// TIA Portal project "APD Gateway Customer Library Source v02_01_00" (V17)
// 00.00.01 - integrated tag tables
// 02.00.01 - v2 will have flat entrypoint
// 02.00.02 - poke ip flattened, next up: finish system parameters
// 02.00.03 - sign formats
// 02.00.04 - line formats
// 02.00.05 - segment formats
// 02.01.00 - released v2

(* hardware
DEVICE "S7-1200 station_1"  S7-1200 Station
   slot 0: "Rack_0"  S7-1200 Rack  Rack  V1.0
   slot 1: "interfacelibrary"  CPU 1215C AC/DC/Rly  6ES7 215-1BG40-0XB0  V4.0
DEVICE "GSD device_1"  GSD.Device.PN
   slot 0: "Rack"  Rack  V1.0
   slot 1: "adpgateway"  Profinet_to_ADP_Gateway  6ES7 212-1AE40-0XB0  V4.5
      slot 0: "Message"  Message
      slot 1: "Interface"  Interface
         slot 1: "Port 1"  Port 1
*)

// ===== PLC "interfacelibrary"  CPU 1215C AC/DC/Rly =====

VAR_GLOBAL   // PLC tag table "Default tag table"
   "System_Byte" AT %MB1 : Byte;
   "FirstScan" AT %M1.0 : Bool;
   "DiagStatusUpdate" AT %M1.1 : Bool;
   "AlwaysTRUE" AT %M1.2 : Bool;
   "AlwaysFALSE" AT %M1.3 : Bool;
   "Clock_Byte" AT %MB0 : Byte;
   "Clock_10Hz" AT %M0.0 : Bool;
   "Clock_5Hz" AT %M0.1 : Bool;
   "Clock_2.5Hz" AT %M0.2 : Bool;
   "Clock_2Hz" AT %M0.3 : Bool;
   "Clock_1.25Hz" AT %M0.4 : Bool;
   "Clock_1Hz" AT %M0.5 : Bool;
   "Clock_0.625Hz" AT %M0.6 : Bool;
   "Clock_0.5Hz" AT %M0.7 : Bool;
END_VAR

VAR_GLOBAL   // PLC tag table "Line Format"
   "Line_0_Font_Size_&_Weight" AT %QB20 : USInt;
   "Line_0_Horizontal_Alignment" AT %QB21 : USInt;
   "Line_1_Font_Size_&_Weight" AT %QB22 : USInt;
   "Line_1_Horizontal_Alignment" AT %QB23 : USInt;
   "Line_2_Font_Size_&_Weight" AT %QB24 : USInt;
   "Line_2_Horizontal_Alignment" AT %QB25 : USInt;
   "Line_3_Font_Size_&_Weight" AT %QB26 : USInt;
   "Line_3_Horizontal_Alignment" AT %QB27 : USInt;
   "Line_4_Font_Size_&_Weight" AT %QB28 : USInt;
   "Line_4_Horizontal_Alignment" AT %QB29 : USInt;
END_VAR

VAR_GLOBAL   // PLC tag table "Segment Format 0"
   "Segment_Format_0_FG_Color" AT %QB50 : SInt;
   "Segment_Format_0_BG_Color" AT %QB51 : SInt;
   "Segment_Format_0_Flash" AT %QB52 : SInt;
   "Segment_Format_0_Line_Number" AT %QB53 : SInt;
   "Segment_Format_0_Text_Byte_0" AT %QB54 : Char;
   "Segment_Format_0_Text_Byte_1" AT %QB55 : Char;
   "Segment_Format_0_Text_Byte_2" AT %QB56 : Char;
   "Segment_Format_0_Text_Byte_3" AT %QB57 : Char;
   "Segment_Format_0_Text_Byte_4" AT %QB58 : Char;
   "Segment_Format_0_Text_Byte_5" AT %QB59 : Char;
   "Segment_Format_0_Text_Byte_6" AT %QB60 : Char;
   "Segment_Format_0_Text_Byte_7" AT %QB61 : Char;
   "Segment_Format_0_Text_Byte_8" AT %QB62 : Char;
   "Segment_Format_0_Text_Byte_9" AT %QB63 : Char;
   "Segment_Format_0_Text_Byte_10" AT %QB64 : Char;
   "Segment_Format_0_Text_Byte_11" AT %QB65 : Char;
   "Segment_Format_0_Text_Byte_12" AT %QB66 : Char;
   "Segment_Format_0_Text_Byte_13" AT %QB67 : Char;
   "Segment_Format_0_Text_Byte_14" AT %QB68 : Char;
   "Segment_Format_0_Text_Byte_15" AT %QB69 : Char;
   "Segment_Format_0_Text_Byte_16" AT %QB70 : Char;
   "Segment_Format_0_Text_Byte_17" AT %QB71 : Char;
   "Segment_Format_0_Text_Byte_18" AT %QB72 : Char;
   "Segment_Format_0_Text_Byte_19" AT %QB73 : Char;
   "Segment_Format_0_Text_Byte_20" AT %QB74 : Char;
   "Segment_Format_0_Text_Byte_21" AT %QB75 : Char;
   "Segment_Format_0_Text_Byte_22" AT %QB76 : Char;
   "Segment_Format_0_Text_Byte_23" AT %QB77 : Char;
   "Segment_Format_0_Text_Byte_24" AT %QB78 : Char;
   "Segment_Format_0_Text_Byte_25" AT %QB79 : Char;
   "Segment_Format_0_Text_Byte_26" AT %QB80 : Char;
   "Segment_Format_0_Text_Byte_27" AT %QB81 : Char;
   "Segment_Format_0_Text_Byte_28" AT %QB82 : Char;
   "Segment_Format_0_Text_Byte_29" AT %QB83 : Char;
   "Segment_Format_0_Text_Byte_30" AT %QB84 : Char;
   "Segment_Format_0_Text_Byte_31" AT %QB85 : Char;
   "Segment_Format_0_Text_Byte_32" AT %QB86 : Char;
   "Segment_Format_0_Text_Byte_33" AT %QB87 : Char;
   "Segment_Format_0_Text_Byte_34" AT %QB88 : Char;
   "Segment_Format_0_Text_Byte_35" AT %QB89 : Char;
   "Segment_Format_0_Text_Byte_36" AT %QB90 : Char;
   "Segment_Format_0_Text_Byte_37" AT %QB91 : Char;
   "Segment_Format_0_Text_Byte_38" AT %QB92 : Char;
   "Segment_Format_0_Text_Byte_39" AT %QB93 : Char;
   "Segment_Format_0_Text_Byte_40" AT %QB94 : Char;
   "Segment_Format_0_Text_Byte_41" AT %QB95 : Char;
   "Segment_Format_0_Text_Byte_42" AT %QB96 : Char;
   "Segment_Format_0_Text_Byte_43" AT %QB97 : Char;
   "Segment_Format_0_Text_Byte_44" AT %QB98 : Char;
   "Segment_Format_0_Text_Byte_45" AT %QB99 : Char;
END_VAR

VAR_GLOBAL   // PLC tag table "Segment Format 1"
   "Segment_Format_1_FG_Color" AT %QB100 : USInt;
   "Segment_Format_1_BG_Color" AT %QB101 : USInt;
   "Segment_Format_1_Flash" AT %QB102 : USInt;
   "Segment_Format_1_Line_Number" AT %QB103 : USInt;
   "Segment_Format_1_Text_Byte_0" AT %QB104 : Char;
   "Segment_Format_1_Text_Byte_1" AT %QB105 : Char;
   "Segment_Format_1_Text_Byte_2" AT %QB106 : Char;
   "Segment_Format_1_Text_Byte_3" AT %QB107 : Char;
   "Segment_Format_1_Text_Byte_4" AT %QB108 : Char;
   "Segment_Format_1_Text_Byte_5" AT %QB109 : Char;
   "Segment_Format_1_Text_Byte_6" AT %QB110 : Char;
   "Segment_Format_1_Text_Byte_7" AT %QB111 : Char;
   "Segment_Format_1_Text_Byte_8" AT %QB112 : Char;
   "Segment_Format_1_Text_Byte_9" AT %QB113 : Char;
   "Segment_Format_1_Text_Byte_10" AT %QB114 : Char;
   "Segment_Format_1_Text_Byte_11" AT %QB115 : Char;
   "Segment_Format_1_Text_Byte_12" AT %QB116 : Char;
   "Segment_Format_1_Text_Byte_13" AT %QB117 : Char;
   "Segment_Format_1_Text_Byte_14" AT %QB118 : Char;
   "Segment_Format_1_Text_Byte_15" AT %QB119 : Char;
   "Segment_Format_1_Text_Byte_16" AT %QB120 : Char;
   "Segment_Format_1_Text_Byte_17" AT %QB121 : Char;
   "Segment_Format_1_Text_Byte_18" AT %QB122 : Char;
   "Segment_Format_1_Text_Byte_19" AT %QB123 : Char;
   "Segment_Format_1_Text_Byte_20" AT %QB124 : Char;
   "Segment_Format_1_Text_Byte_21" AT %QB125 : Char;
   "Segment_Format_1_Text_Byte_22" AT %QB126 : Char;
   "Segment_Format_1_Text_Byte_23" AT %QB127 : Char;
   "Segment_Format_1_Text_Byte_24" AT %QB128 : Char;
   "Segment_Format_1_Text_Byte_25" AT %QB129 : Char;
   "Segment_Format_1_Text_Byte_26" AT %QB130 : Char;
   "Segment_Format_1_Text_Byte_27" AT %QB131 : Char;
   "Segment_Format_1_Text_Byte_28" AT %QB132 : Char;
   "Segment_Format_1_Text_Byte_29" AT %QB133 : Char;
   "Segment_Format_1_Text_Byte_30" AT %QB134 : Char;
   "Segment_Format_1_Text_Byte_31" AT %QB135 : Char;
   "Segment_Format_1_Text_Byte_32" AT %QB136 : Char;
   "Segment_Format_1_Text_Byte_33" AT %QB137 : Char;
   "Segment_Format_1_Text_Byte_34" AT %QB138 : Char;
   "Segment_Format_1_Text_Byte_35" AT %QB139 : Char;
   "Segment_Format_1_Text_Byte_36" AT %QB140 : Char;
   "Segment_Format_1_Text_Byte_37" AT %QB141 : Char;
   "Segment_Format_1_Text_Byte_38" AT %QB142 : Char;
   "Segment_Format_1_Text_Byte_39" AT %QB143 : Char;
   "Segment_Format_1_Text_Byte_40" AT %QB144 : Char;
   "Segment_Format_1_Text_Byte_41" AT %QB145 : Char;
   "Segment_Format_1_Text_Byte_42" AT %QB146 : Char;
   "Segment_Format_1_Text_Byte_43" AT %QB147 : Char;
   "Segment_Format_1_Text_Byte_44" AT %QB148 : Char;
   "Segment_Format_1_Text_Byte_45" AT %QB149 : Char;
END_VAR

VAR_GLOBAL   // PLC tag table "Segment Format 2"
   "Segment_Format_2_FG_Color" AT %QB150 : USInt;
   "Segment_Format_2_BG_Color" AT %QB151 : USInt;
   "Segment_Format_2_Flash" AT %QB152 : USInt;
   "Segment_Format_2_Line_Number" AT %QB153 : USInt;
   "Segment_Format_2_Text_Byte_0" AT %QB154 : Char;
   "Segment_Format_2_Text_Byte_1" AT %QB155 : Char;
   "Segment_Format_2_Text_Byte_2" AT %QB156 : Char;
   "Segment_Format_2_Text_Byte_3" AT %QB157 : Char;
   "Segment_Format_2_Text_Byte_4" AT %QB158 : Char;
   "Segment_Format_2_Text_Byte_5" AT %QB159 : Char;
   "Segment_Format_2_Text_Byte_6" AT %QB160 : Char;
   "Segment_Format_2_Text_Byte_7" AT %QB161 : Char;
   "Segment_Format_2_Text_Byte_8" AT %QB162 : Char;
   "Segment_Format_2_Text_Byte_9" AT %QB163 : Char;
   "Segment_Format_2_Text_Byte_10" AT %QB164 : Char;
   "Segment_Format_2_Text_Byte_11" AT %QB165 : Char;
   "Segment_Format_2_Text_Byte_12" AT %QB166 : Char;
   "Segment_Format_2_Text_Byte_13" AT %QB167 : Char;
   "Segment_Format_2_Text_Byte_14" AT %QB168 : Char;
   "Segment_Format_2_Text_Byte_15" AT %QB169 : Char;
   "Segment_Format_2_Text_Byte_16" AT %QB170 : Char;
   "Segment_Format_2_Text_Byte_17" AT %QB171 : Char;
   "Segment_Format_2_Text_Byte_18" AT %QB172 : Char;
   "Segment_Format_2_Text_Byte_19" AT %QB173 : Char;
   "Segment_Format_2_Text_Byte_20" AT %QB174 : Char;
   "Segment_Format_2_Text_Byte_21" AT %QB175 : Char;
   "Segment_Format_2_Text_Byte_22" AT %QB176 : Char;
   "Segment_Format_2_Text_Byte_23" AT %QB177 : Char;
   "Segment_Format_2_Text_Byte_24" AT %QB178 : Char;
   "Segment_Format_2_Text_Byte_25" AT %QB179 : Char;
   "Segment_Format_2_Text_Byte_26" AT %QB180 : Char;
   "Segment_Format_2_Text_Byte_27" AT %QB181 : Char;
   "Segment_Format_2_Text_Byte_28" AT %QB182 : Char;
   "Segment_Format_2_Text_Byte_29" AT %QB183 : Char;
   "Segment_Format_2_Text_Byte_30" AT %QB184 : Char;
   "Segment_Format_2_Text_Byte_31" AT %QB185 : Char;
   "Segment_Format_2_Text_Byte_32" AT %QB186 : Char;
   "Segment_Format_2_Text_Byte_33" AT %QB187 : Char;
   "Segment_Format_2_Text_Byte_34" AT %QB188 : Char;
   "Segment_Format_2_Text_Byte_35" AT %QB189 : Char;
   "Segment_Format_2_Text_Byte_36" AT %QB190 : Char;
   "Segment_Format_2_Text_Byte_37" AT %QB191 : Char;
   "Segment_Format_2_Text_Byte_38" AT %QB192 : Char;
   "Segment_Format_2_Text_Byte_39" AT %QB193 : Char;
   "Segment_Format_2_Text_Byte_40" AT %QB194 : Char;
   "Segment_Format_2_Text_Byte_41" AT %QB195 : Char;
   "Segment_Format_2_Text_Byte_42" AT %QB196 : Char;
   "Segment_Format_2_Text_Byte_43" AT %QB197 : Char;
   "Segment_Format_2_Text_Byte_44" AT %QB198 : Char;
   "Segment_Format_2_Text_Byte_45" AT %QB199 : Char;
END_VAR

VAR_GLOBAL   // PLC tag table "Segment Format 3"
   "Segment_Format_3_FG_Color" AT %QB200 : USInt;
   "Segment_Format_3_BG_Color" AT %QB201 : USInt;
   "Segment_Format_3_Flash" AT %QB202 : USInt;
   "Segment_Format_3_Line_Number" AT %QB203 : USInt;
   "Segment_Format_3_Text_Byte_0" AT %QB204 : Char;
   "Segment_Format_3_Text_Byte_1" AT %QB205 : Char;
   "Segment_Format_3_Text_Byte_2" AT %QB206 : Char;
   "Segment_Format_3_Text_Byte_3" AT %QB207 : Char;
   "Segment_Format_3_Text_Byte_4" AT %QB208 : Char;
   "Segment_Format_3_Text_Byte_5" AT %QB209 : Char;
   "Segment_Format_3_Text_Byte_6" AT %QB210 : Char;
   "Segment_Format_3_Text_Byte_7" AT %QB211 : Char;
   "Segment_Format_3_Text_Byte_8" AT %QB212 : Char;
   "Segment_Format_3_Text_Byte_9" AT %QB213 : Char;
   "Segment_Format_3_Text_Byte_10" AT %QB214 : Char;
   "Segment_Format_3_Text_Byte_11" AT %QB215 : Char;
   "Segment_Format_3_Text_Byte_12" AT %QB216 : Char;
   "Segment_Format_3_Text_Byte_13" AT %QB217 : Char;
   "Segment_Format_3_Text_Byte_14" AT %QB218 : Char;
   "Segment_Format_3_Text_Byte_15" AT %QB219 : Char;
   "Segment_Format_3_Text_Byte_16" AT %QB220 : Char;
   "Segment_Format_3_Text_Byte_17" AT %QB221 : Char;
   "Segment_Format_3_Text_Byte_18" AT %QB222 : Char;
   "Segment_Format_3_Text_Byte_19" AT %QB223 : Char;
   "Segment_Format_3_Text_Byte_20" AT %QB224 : Char;
   "Segment_Format_3_Text_Byte_21" AT %QB225 : Char;
   "Segment_Format_3_Text_Byte_22" AT %QB226 : Char;
   "Segment_Format_3_Text_Byte_23" AT %QB227 : Char;
   "Segment_Format_3_Text_Byte_24" AT %QB228 : Char;
   "Segment_Format_3_Text_Byte_25" AT %QB229 : Char;
   "Segment_Format_3_Text_Byte_26" AT %QB230 : Char;
   "Segment_Format_3_Text_Byte_27" AT %QB231 : Char;
   "Segment_Format_3_Text_Byte_28" AT %QB232 : Char;
   "Segment_Format_3_Text_Byte_29" AT %QB233 : Char;
   "Segment_Format_3_Text_Byte_30" AT %QB234 : Char;
   "Segment_Format_3_Text_Byte_31" AT %QB235 : Char;
   "Segment_Format_3_Text_Byte_32" AT %QB236 : Char;
   "Segment_Format_3_Text_Byte_33" AT %QB237 : Char;
   "Segment_Format_3_Text_Byte_34" AT %QB238 : Char;
   "Segment_Format_3_Text_Byte_35" AT %QB239 : Char;
   "Segment_Format_3_Text_Byte_36" AT %QB240 : Char;
   "Segment_Format_3_Text_Byte_37" AT %QB241 : Char;
   "Segment_Format_3_Text_Byte_38" AT %QB242 : Char;
   "Segment_Format_3_Text_Byte_39" AT %QB243 : Char;
   "Segment_Format_3_Text_Byte_40" AT %QB244 : Char;
   "Segment_Format_3_Text_Byte_41" AT %QB245 : Char;
   "Segment_Format_3_Text_Byte_42" AT %QB246 : Char;
   "Segment_Format_3_Text_Byte_43" AT %QB247 : Char;
   "Segment_Format_3_Text_Byte_44" AT %QB248 : Char;
   "Segment_Format_3_Text_Byte_45" AT %QB249 : Char;
END_VAR

VAR_GLOBAL   // PLC tag table "Segment Format 4"
   "Segment_Format_4_FG_Color" AT %QB250 : USInt;
   "Segment_Format_4_BG_Color" AT %QB251 : USInt;
   "Segment_Format_4_Flash" AT %QB252 : USInt;
   "Segment_Format_4_Line_Number" AT %QB253 : USInt;
   "Segment_Format_4_Text_Byte_0" AT %QB254 : Char;
   "Segment_Format_4_Text_Byte_1" AT %QB255 : Char;
   "Segment_Format_4_Text_Byte_2" AT %QB256 : Char;
   "Segment_Format_4_Text_Byte_3" AT %QB257 : Char;
   "Segment_Format_4_Text_Byte_4" AT %QB258 : Char;
   "Segment_Format_4_Text_Byte_5" AT %QB259 : Char;
   "Segment_Format_4_Text_Byte_6" AT %QB260 : Char;
   "Segment_Format_4_Text_Byte_7" AT %QB261 : Char;
   "Segment_Format_4_Text_Byte_8" AT %QB262 : Char;
   "Segment_Format_4_Text_Byte_9" AT %QB263 : Char;
   "Segment_Format_4_Text_Byte_10" AT %QB264 : Char;
   "Segment_Format_4_Text_Byte_11" AT %QB265 : Char;
   "Segment_Format_4_Text_Byte_12" AT %QB266 : Char;
   "Segment_Format_4_Text_Byte_13" AT %QB267 : Char;
   "Segment_Format_4_Text_Byte_14" AT %QB268 : Char;
   "Segment_Format_4_Text_Byte_15" AT %QB269 : Char;
   "Segment_Format_4_Text_Byte_16" AT %QB270 : Char;
   "Segment_Format_4_Text_Byte_17" AT %QB271 : Char;
   "Segment_Format_4_Text_Byte_18" AT %QB272 : Char;
   "Segment_Format_4_Text_Byte_19" AT %QB273 : Char;
   "Segment_Format_4_Text_Byte_20" AT %QB274 : Char;
   "Segment_Format_4_Text_Byte_21" AT %QB275 : Char;
   "Segment_Format_4_Text_Byte_22" AT %QB276 : Char;
   "Segment_Format_4_Text_Byte_23" AT %QB277 : Char;
   "Segment_Format_4_Text_Byte_24" AT %QB278 : Char;
   "Segment_Format_4_Text_Byte_25" AT %QB279 : Char;
   "Segment_Format_4_Text_Byte_26" AT %QB280 : Char;
   "Segment_Format_4_Text_Byte_27" AT %QB281 : Char;
   "Segment_Format_4_Text_Byte_28" AT %QB282 : Char;
   "Segment_Format_4_Text_Byte_29" AT %QB283 : Char;
   "Segment_Format_4_Text_Byte_30" AT %QB284 : Char;
   "Segment_Format_4_Text_Byte_31" AT %QB285 : Char;
   "Segment_Format_4_Text_Byte_32" AT %QB286 : Char;
   "Segment_Format_4_Text_Byte_33" AT %QB287 : Char;
   "Segment_Format_4_Text_Byte_34" AT %QB288 : Char;
   "Segment_Format_4_Text_Byte_35" AT %QB289 : Char;
   "Segment_Format_4_Text_Byte_36" AT %QB290 : Char;
   "Segment_Format_4_Text_Byte_37" AT %QB291 : Char;
   "Segment_Format_4_Text_Byte_38" AT %QB292 : Char;
   "Segment_Format_4_Text_Byte_39" AT %QB293 : Char;
   "Segment_Format_4_Text_Byte_40" AT %QB294 : Char;
   "Segment_Format_4_Text_Byte_41" AT %QB295 : Char;
   "Segment_Format_4_Text_Byte_42" AT %QB296 : Char;
   "Segment_Format_4_Text_Byte_43" AT %QB297 : Char;
   "Segment_Format_4_Text_Byte_44" AT %QB298 : Char;
   "Segment_Format_4_Text_Byte_45" AT %QB299 : Char;
END_VAR

VAR_GLOBAL   // PLC tag table "Segment Format 5"
   "Segment_Format_5_FG_Color" AT %QB300 : USInt;
   "Segment_Format_5_BG_Color" AT %QB301 : USInt;
   "Segment_Format_5_Flash" AT %QB302 : USInt;
   "Segment_Format_5_Line_Number" AT %QB303 : USInt;
   "Segment_Format_5_Text_Byte_0" AT %QB304 : Char;
   "Segment_Format_5_Text_Byte_1" AT %QB305 : Char;
   "Segment_Format_5_Text_Byte_2" AT %QB306 : Char;
   "Segment_Format_5_Text_Byte_3" AT %QB307 : Char;
   "Segment_Format_5_Text_Byte_4" AT %QB308 : Char;
   "Segment_Format_5_Text_Byte_5" AT %QB309 : Char;
   "Segment_Format_5_Text_Byte_6" AT %QB310 : Char;
   "Segment_Format_5_Text_Byte_7" AT %QB311 : Char;
   "Segment_Format_5_Text_Byte_8" AT %QB312 : Char;
   "Segment_Format_5_Text_Byte_9" AT %QB313 : Char;
   "Segment_Format_5_Text_Byte_10" AT %QB314 : Char;
   "Segment_Format_5_Text_Byte_11" AT %QB315 : Char;
   "Segment_Format_5_Text_Byte_12" AT %QB316 : Char;
   "Segment_Format_5_Text_Byte_13" AT %QB317 : Char;
   "Segment_Format_5_Text_Byte_14" AT %QB318 : Char;
   "Segment_Format_5_Text_Byte_15" AT %QB319 : Char;
   "Segment_Format_5_Text_Byte_16" AT %QB320 : Char;
   "Segment_Format_5_Text_Byte_17" AT %QB321 : Char;
   "Segment_Format_5_Text_Byte_18" AT %QB322 : Char;
   "Segment_Format_5_Text_Byte_19" AT %QB323 : Char;
   "Segment_Format_5_Text_Byte_20" AT %QB324 : Char;
   "Segment_Format_5_Text_Byte_21" AT %QB325 : Char;
   "Segment_Format_5_Text_Byte_22" AT %QB326 : Char;
   "Segment_Format_5_Text_Byte_23" AT %QB327 : Char;
   "Segment_Format_5_Text_Byte_24" AT %QB328 : Char;
   "Segment_Format_5_Text_Byte_25" AT %QB329 : Char;
   "Segment_Format_5_Text_Byte_26" AT %QB330 : Char;
   "Segment_Format_5_Text_Byte_27" AT %QB331 : Char;
   "Segment_Format_5_Text_Byte_28" AT %QB332 : Char;
   "Segment_Format_5_Text_Byte_29" AT %QB333 : Char;
   "Segment_Format_5_Text_Byte_30" AT %QB334 : Char;
   "Segment_Format_5_Text_Byte_31" AT %QB335 : Char;
   "Segment_Format_5_Text_Byte_32" AT %QB336 : Char;
   "Segment_Format_5_Text_Byte_33" AT %QB337 : Char;
   "Segment_Format_5_Text_Byte_34" AT %QB338 : Char;
   "Segment_Format_5_Text_Byte_35" AT %QB339 : Char;
   "Segment_Format_5_Text_Byte_36" AT %QB340 : Char;
   "Segment_Format_5_Text_Byte_37" AT %QB341 : Char;
   "Segment_Format_5_Text_Byte_38" AT %QB342 : Char;
   "Segment_Format_5_Text_Byte_39" AT %QB343 : Char;
   "Segment_Format_5_Text_Byte_40" AT %QB344 : Char;
   "Segment_Format_5_Text_Byte_41" AT %QB345 : Char;
   "Segment_Format_5_Text_Byte_42" AT %QB346 : Char;
   "Segment_Format_5_Text_Byte_43" AT %QB347 : Char;
   "Segment_Format_5_Text_Byte_44" AT %QB348 : Char;
   "Segment_Format_5_Text_Byte_45" AT %QB349 : Char;
END_VAR

VAR_GLOBAL   // PLC tag table "Segment Format 6"
   "Segment_Format_6_FG_Color" AT %QB350 : USInt;
   "Segment_Format_6_BG_Color" AT %QB351 : USInt;
   "Segment_Format_6_Flash" AT %QB352 : USInt;
   "Segment_Format_6_Line_Number" AT %QB353 : USInt;
   "Segment_Format_6_Text_Byte_0" AT %QB354 : Char;
   "Segment_Format_6_Text_Byte_1" AT %QB355 : Char;
   "Segment_Format_6_Text_Byte_2" AT %QB356 : Char;
   "Segment_Format_6_Text_Byte_3" AT %QB357 : Char;
   "Segment_Format_6_Text_Byte_4" AT %QB358 : Char;
   "Segment_Format_6_Text_Byte_5" AT %QB359 : Char;
   "Segment_Format_6_Text_Byte_6" AT %QB360 : Char;
   "Segment_Format_6_Text_Byte_7" AT %QB361 : Char;
   "Segment_Format_6_Text_Byte_8" AT %QB362 : Char;
   "Segment_Format_6_Text_Byte_9" AT %QB363 : Char;
   "Segment_Format_6_Text_Byte_10" AT %QB364 : Char;
   "Segment_Format_6_Text_Byte_11" AT %QB365 : Char;
   "Segment_Format_6_Text_Byte_12" AT %QB366 : Char;
   "Segment_Format_6_Text_Byte_13" AT %QB367 : Char;
   "Segment_Format_6_Text_Byte_14" AT %QB368 : Char;
   "Segment_Format_6_Text_Byte_15" AT %QB369 : Char;
   "Segment_Format_6_Text_Byte_16" AT %QB370 : Char;
   "Segment_Format_6_Text_Byte_17" AT %QB371 : Char;
   "Segment_Format_6_Text_Byte_18" AT %QB372 : Char;
   "Segment_Format_6_Text_Byte_19" AT %QB373 : Char;
   "Segment_Format_6_Text_Byte_20" AT %QB374 : Char;
   "Segment_Format_6_Text_Byte_21" AT %QB375 : Char;
   "Segment_Format_6_Text_Byte_22" AT %QB376 : Char;
   "Segment_Format_6_Text_Byte_23" AT %QB377 : Char;
   "Segment_Format_6_Text_Byte_24" AT %QB378 : Char;
   "Segment_Format_6_Text_Byte_25" AT %QB379 : Char;
   "Segment_Format_6_Text_Byte_26" AT %QB380 : Char;
   "Segment_Format_6_Text_Byte_27" AT %QB381 : Char;
   "Segment_Format_6_Text_Byte_28" AT %QB382 : Char;
   "Segment_Format_6_Text_Byte_29" AT %QB383 : Char;
   "Segment_Format_6_Text_Byte_30" AT %QB384 : Char;
   "Segment_Format_6_Text_Byte_31" AT %QB385 : Char;
   "Segment_Format_6_Text_Byte_32" AT %QB386 : Char;
   "Segment_Format_6_Text_Byte_33" AT %QB387 : Char;
   "Segment_Format_6_Text_Byte_34" AT %QB388 : Char;
   "Segment_Format_6_Text_Byte_35" AT %QB389 : Char;
   "Segment_Format_6_Text_Byte_36" AT %QB390 : Char;
   "Segment_Format_6_Text_Byte_37" AT %QB391 : Char;
   "Segment_Format_6_Text_Byte_38" AT %QB392 : Char;
   "Segment_Format_6_Text_Byte_39" AT %QB393 : Char;
   "Segment_Format_6_Text_Byte_40" AT %QB394 : Char;
   "Segment_Format_6_Text_Byte_41" AT %QB395 : Char;
   "Segment_Format_6_Text_Byte_42" AT %QB396 : Char;
   "Segment_Format_6_Text_Byte_43" AT %QB397 : Char;
   "Segment_Format_6_Text_Byte_44" AT %QB398 : Char;
   "Segment_Format_6_Text_Byte_45" AT %QB399 : Char;
END_VAR

VAR_GLOBAL   // PLC tag table "Segment Format 7"
   "Segment_Format_7_FG_Color" AT %QB400 : USInt;
   "Segment_Format_7_BG_Color" AT %QB401 : USInt;
   "Segment_Format_7_Flash" AT %QB402 : USInt;
   "Segment_Format_7_Line_Number" AT %QB403 : USInt;
   "Segment_Format_7_Text_Byte_0" AT %QB404 : Char;
   "Segment_Format_7_Text_Byte_1" AT %QB405 : Char;
   "Segment_Format_7_Text_Byte_2" AT %QB406 : Char;
   "Segment_Format_7_Text_Byte_3" AT %QB407 : Char;
   "Segment_Format_7_Text_Byte_4" AT %QB408 : Char;
   "Segment_Format_7_Text_Byte_5" AT %QB409 : Char;
   "Segment_Format_7_Text_Byte_6" AT %QB410 : Char;
   "Segment_Format_7_Text_Byte_7" AT %QB411 : Char;
   "Segment_Format_7_Text_Byte_8" AT %QB412 : Char;
   "Segment_Format_7_Text_Byte_9" AT %QB413 : Char;
   "Segment_Format_7_Text_Byte_10" AT %QB414 : Char;
   "Segment_Format_7_Text_Byte_11" AT %QB415 : Char;
   "Segment_Format_7_Text_Byte_12" AT %QB416 : Char;
   "Segment_Format_7_Text_Byte_13" AT %QB417 : Char;
   "Segment_Format_7_Text_Byte_14" AT %QB418 : Char;
   "Segment_Format_7_Text_Byte_15" AT %QB419 : Char;
   "Segment_Format_7_Text_Byte_16" AT %QB420 : Char;
   "Segment_Format_7_Text_Byte_17" AT %QB421 : Char;
   "Segment_Format_7_Text_Byte_18" AT %QB422 : Char;
   "Segment_Format_7_Text_Byte_19" AT %QB423 : Char;
   "Segment_Format_7_Text_Byte_20" AT %QB424 : Char;
   "Segment_Format_7_Text_Byte_21" AT %QB425 : Char;
   "Segment_Format_7_Text_Byte_22" AT %QB426 : Char;
   "Segment_Format_7_Text_Byte_23" AT %QB427 : Char;
   "Segment_Format_7_Text_Byte_24" AT %QB428 : Char;
   "Segment_Format_7_Text_Byte_25" AT %QB429 : Char;
   "Segment_Format_7_Text_Byte_26" AT %QB430 : Char;
   "Segment_Format_7_Text_Byte_27" AT %QB431 : Char;
   "Segment_Format_7_Text_Byte_28" AT %QB432 : Char;
   "Segment_Format_7_Text_Byte_29" AT %QB433 : Char;
   "Segment_Format_7_Text_Byte_30" AT %QB434 : Char;
   "Segment_Format_7_Text_Byte_31" AT %QB435 : Char;
   "Segment_Format_7_Text_Byte_32" AT %QB436 : Char;
   "Segment_Format_7_Text_Byte_33" AT %QB437 : Char;
   "Segment_Format_7_Text_Byte_34" AT %QB438 : Char;
   "Segment_Format_7_Text_Byte_35" AT %QB439 : Char;
   "Segment_Format_7_Text_Byte_36" AT %QB440 : Char;
   "Segment_Format_7_Text_Byte_37" AT %QB441 : Char;
   "Segment_Format_7_Text_Byte_38" AT %QB442 : Char;
   "Segment_Format_7_Text_Byte_39" AT %QB443 : Char;
   "Segment_Format_7_Text_Byte_40" AT %QB444 : Char;
   "Segment_Format_7_Text_Byte_41" AT %QB445 : Char;
   "Segment_Format_7_Text_Byte_42" AT %QB446 : Char;
   "Segment_Format_7_Text_Byte_43" AT %QB447 : Char;
   "Segment_Format_7_Text_Byte_44" AT %QB448 : Char;
   "Segment_Format_7_Text_Byte_45" AT %QB449 : Char;
END_VAR

VAR_GLOBAL   // PLC tag table "Segment Format 8"
   "Segment_Format_8_FG_Color" AT %QB450 : USInt;
   "Segment_Format_8_BG_Color" AT %QB451 : USInt;
   "Segment_Format_8_Flash" AT %QB452 : USInt;
   "Segment_Format_8_Line_Number" AT %QB453 : USInt;
   "Segment_Format_8_Text_Byte_0" AT %QB454 : Char;
   "Segment_Format_8_Text_Byte_1" AT %QB455 : Char;
   "Segment_Format_8_Text_Byte_2" AT %QB456 : Char;
   "Segment_Format_8_Text_Byte_3" AT %QB457 : Char;
   "Segment_Format_8_Text_Byte_4" AT %QB458 : Char;
   "Segment_Format_8_Text_Byte_5" AT %QB459 : Char;
   "Segment_Format_8_Text_Byte_6" AT %QB460 : Char;
   "Segment_Format_8_Text_Byte_7" AT %QB461 : Char;
   "Segment_Format_8_Text_Byte_8" AT %QB462 : Char;
   "Segment_Format_8_Text_Byte_9" AT %QB463 : Char;
   "Segment_Format_8_Text_Byte_10" AT %QB464 : Char;
   "Segment_Format_8_Text_Byte_11" AT %QB465 : Char;
   "Segment_Format_8_Text_Byte_12" AT %QB466 : Char;
   "Segment_Format_8_Text_Byte_13" AT %QB467 : Char;
   "Segment_Format_8_Text_Byte_14" AT %QB468 : Char;
   "Segment_Format_8_Text_Byte_15" AT %QB469 : Char;
   "Segment_Format_8_Text_Byte_16" AT %QB470 : Char;
   "Segment_Format_8_Text_Byte_17" AT %QB471 : Char;
   "Segment_Format_8_Text_Byte_18" AT %QB472 : Char;
   "Segment_Format_8_Text_Byte_19" AT %QB473 : Char;
   "Segment_Format_8_Text_Byte_20" AT %QB474 : Char;
   "Segment_Format_8_Text_Byte_21" AT %QB475 : Char;
   "Segment_Format_8_Text_Byte_22" AT %QB476 : Char;
   "Segment_Format_8_Text_Byte_23" AT %QB477 : Char;
   "Segment_Format_8_Text_Byte_24" AT %QB478 : Char;
   "Segment_Format_8_Text_Byte_25" AT %QB479 : Char;
   "Segment_Format_8_Text_Byte_26" AT %QB480 : Char;
   "Segment_Format_8_Text_Byte_27" AT %QB481 : Char;
   "Segment_Format_8_Text_Byte_28" AT %QB482 : Char;
   "Segment_Format_8_Text_Byte_29" AT %QB483 : Char;
   "Segment_Format_8_Text_Byte_30" AT %QB484 : Char;
   "Segment_Format_8_Text_Byte_31" AT %QB485 : Char;
   "Segment_Format_8_Text_Byte_32" AT %QB486 : Char;
   "Segment_Format_8_Text_Byte_33" AT %QB487 : Char;
   "Segment_Format_8_Text_Byte_34" AT %QB488 : Char;
   "Segment_Format_8_Text_Byte_35" AT %QB489 : Char;
   "Segment_Format_8_Text_Byte_36" AT %QB490 : Char;
   "Segment_Format_8_Text_Byte_37" AT %QB491 : Char;
   "Segment_Format_8_Text_Byte_38" AT %QB492 : Char;
   "Segment_Format_8_Text_Byte_39" AT %QB493 : Char;
   "Segment_Format_8_Text_Byte_40" AT %QB494 : Char;
   "Segment_Format_8_Text_Byte_41" AT %QB495 : Char;
   "Segment_Format_8_Text_Byte_42" AT %QB496 : Char;
   "Segment_Format_8_Text_Byte_43" AT %QB497 : Char;
   "Segment_Format_8_Text_Byte_44" AT %QB498 : Char;
   "Segment_Format_8_Text_Byte_45" AT %QB499 : Char;
END_VAR

VAR_GLOBAL   // PLC tag table "Segment Format 9"
   "Segment_Format_9_FG_Color" AT %QB500 : USInt;
   "Segment_Format_9_BG_Color" AT %QB501 : USInt;
   "Segment_Format_9_Flash" AT %QB502 : USInt;
   "Segment_Format_9_Line_Number" AT %QB503 : USInt;
   "Segment_Format_9_Text_Byte_0" AT %QB504 : Char;
   "Segment_Format_9_Text_Byte_1" AT %QB505 : Char;
   "Segment_Format_9_Text_Byte_2" AT %QB506 : Char;
   "Segment_Format_9_Text_Byte_3" AT %QB507 : Char;
   "Segment_Format_9_Text_Byte_4" AT %QB508 : Char;
   "Segment_Format_9_Text_Byte_5" AT %QB509 : Char;
   "Segment_Format_9_Text_Byte_6" AT %QB510 : Char;
   "Segment_Format_9_Text_Byte_7" AT %QB511 : Char;
   "Segment_Format_9_Text_Byte_8" AT %QB512 : Char;
   "Segment_Format_9_Text_Byte_9" AT %QB513 : Char;
   "Segment_Format_9_Text_Byte_10" AT %QB514 : Char;
   "Segment_Format_9_Text_Byte_11" AT %QB515 : Char;
   "Segment_Format_9_Text_Byte_12" AT %QB516 : Char;
   "Segment_Format_9_Text_Byte_13" AT %QB517 : Char;
   "Segment_Format_9_Text_Byte_14" AT %QB518 : Char;
   "Segment_Format_9_Text_Byte_15" AT %QB519 : Char;
   "Segment_Format_9_Text_Byte_16" AT %QB520 : Char;
   "Segment_Format_9_Text_Byte_17" AT %QB521 : Char;
   "Segment_Format_9_Text_Byte_18" AT %QB522 : Char;
   "Segment_Format_9_Text_Byte_19" AT %QB523 : Char;
   "Segment_Format_9_Text_Byte_20" AT %QB524 : Char;
   "Segment_Format_9_Text_Byte_21" AT %QB525 : Char;
   "Segment_Format_9_Text_Byte_22" AT %QB526 : Char;
   "Segment_Format_9_Text_Byte_23" AT %QB527 : Char;
   "Segment_Format_9_Text_Byte_24" AT %QB528 : Char;
   "Segment_Format_9_Text_Byte_25" AT %QB529 : Char;
   "Segment_Format_9_Text_Byte_26" AT %QB530 : Char;
   "Segment_Format_9_Text_Byte_27" AT %QB531 : Char;
   "Segment_Format_9_Text_Byte_28" AT %QB532 : Char;
   "Segment_Format_9_Text_Byte_29" AT %QB533 : Char;
   "Segment_Format_9_Text_Byte_30" AT %QB534 : Char;
   "Segment_Format_9_Text_Byte_31" AT %QB535 : Char;
   "Segment_Format_9_Text_Byte_32" AT %QB536 : Char;
   "Segment_Format_9_Text_Byte_33" AT %QB537 : Char;
   "Segment_Format_9_Text_Byte_34" AT %QB538 : Char;
   "Segment_Format_9_Text_Byte_35" AT %QB539 : Char;
   "Segment_Format_9_Text_Byte_36" AT %QB540 : Char;
   "Segment_Format_9_Text_Byte_37" AT %QB541 : Char;
   "Segment_Format_9_Text_Byte_38" AT %QB542 : Char;
   "Segment_Format_9_Text_Byte_39" AT %QB543 : Char;
   "Segment_Format_9_Text_Byte_40" AT %QB544 : Char;
   "Segment_Format_9_Text_Byte_41" AT %QB545 : Char;
   "Segment_Format_9_Text_Byte_42" AT %QB546 : Char;
   "Segment_Format_9_Text_Byte_43" AT %QB547 : Char;
   "Segment_Format_9_Text_Byte_44" AT %QB548 : Char;
   "Segment_Format_9_Text_Byte_45" AT %QB549 : Char;
END_VAR

VAR_GLOBAL   // PLC tag table "Segment Format 10"
   "Segment_Format_10_FG_Color" AT %QB550 : USInt;
   "Segment_Format_10_BG_Color" AT %QB551 : USInt;
   "Segment_Format_10_Flash" AT %QB552 : USInt;
   "Segment_Format_10_Line_Number" AT %QB553 : USInt;
   "Segment_Format_10_Text_Byte_0" AT %QB554 : Char;
   "Segment_Format_10_Text_Byte_1" AT %QB555 : Char;
   "Segment_Format_10_Text_Byte_2" AT %QB556 : Char;
   "Segment_Format_10_Text_Byte_3" AT %QB557 : Char;
   "Segment_Format_10_Text_Byte_4" AT %QB558 : Char;
   "Segment_Format_10_Text_Byte_5" AT %QB559 : Char;
   "Segment_Format_10_Text_Byte_6" AT %QB560 : Char;
   "Segment_Format_10_Text_Byte_7" AT %QB561 : Char;
   "Segment_Format_10_Text_Byte_8" AT %QB562 : Char;
   "Segment_Format_10_Text_Byte_9" AT %QB563 : Char;
   "Segment_Format_10_Text_Byte_10" AT %QB564 : Char;
   "Segment_Format_10_Text_Byte_11" AT %QB565 : Char;
   "Segment_Format_10_Text_Byte_12" AT %QB566 : Char;
   "Segment_Format_10_Text_Byte_13" AT %QB567 : Char;
   "Segment_Format_10_Text_Byte_14" AT %QB568 : Char;
   "Segment_Format_10_Text_Byte_15" AT %QB569 : Char;
   "Segment_Format_10_Text_Byte_16" AT %QB570 : Char;
   "Segment_Format_10_Text_Byte_17" AT %QB571 : Char;
   "Segment_Format_10_Text_Byte_18" AT %QB572 : Char;
   "Segment_Format_10_Text_Byte_19" AT %QB573 : Char;
   "Segment_Format_10_Text_Byte_20" AT %QB574 : Char;
   "Segment_Format_10_Text_Byte_21" AT %QB575 : Char;
   "Segment_Format_10_Text_Byte_22" AT %QB576 : Char;
   "Segment_Format_10_Text_Byte_23" AT %QB577 : Char;
   "Segment_Format_10_Text_Byte_24" AT %QB578 : Char;
   "Segment_Format_10_Text_Byte_25" AT %QB579 : Char;
   "Segment_Format_10_Text_Byte_26" AT %QB580 : Char;
   "Segment_Format_10_Text_Byte_27" AT %QB581 : Char;
   "Segment_Format_10_Text_Byte_28" AT %QB582 : Char;
   "Segment_Format_10_Text_Byte_29" AT %QB583 : Char;
   "Segment_Format_10_Text_Byte_30" AT %QB584 : Char;
   "Segment_Format_10_Text_Byte_31" AT %QB585 : Char;
   "Segment_Format_10_Text_Byte_32" AT %QB586 : Char;
   "Segment_Format_10_Text_Byte_33" AT %QB587 : Char;
   "Segment_Format_10_Text_Byte_34" AT %QB588 : Char;
   "Segment_Format_10_Text_Byte_35" AT %QB589 : Char;
   "Segment_Format_10_Text_Byte_36" AT %QB590 : Char;
   "Segment_Format_10_Text_Byte_37" AT %QB591 : Char;
   "Segment_Format_10_Text_Byte_38" AT %QB592 : Char;
   "Segment_Format_10_Text_Byte_39" AT %QB593 : Char;
   "Segment_Format_10_Text_Byte_40" AT %QB594 : Char;
   "Segment_Format_10_Text_Byte_41" AT %QB595 : Char;
   "Segment_Format_10_Text_Byte_42" AT %QB596 : Char;
   "Segment_Format_10_Text_Byte_43" AT %QB597 : Char;
   "Segment_Format_10_Text_Byte_44" AT %QB598 : Char;
   "Segment_Format_10_Text_Byte_45" AT %QB599 : Char;
END_VAR

VAR_GLOBAL   // PLC tag table "Segment Format 11"
   "Segment_Format_11_FG_Color" AT %QB600 : USInt;
   "Segment_Format_11_BG_Color" AT %QB601 : USInt;
   "Segment_Format_11_Flash" AT %QB602 : USInt;
   "Segment_Format_11_Line_Number" AT %QB603 : USInt;
   "Segment_Format_11_Text_Byte_0" AT %QB604 : Char;
   "Segment_Format_11_Text_Byte_1" AT %QB605 : Char;
   "Segment_Format_11_Text_Byte_2" AT %QB606 : Char;
   "Segment_Format_11_Text_Byte_3" AT %QB607 : Char;
   "Segment_Format_11_Text_Byte_4" AT %QB608 : Char;
   "Segment_Format_11_Text_Byte_5" AT %QB609 : Char;
   "Segment_Format_11_Text_Byte_6" AT %QB610 : Char;
   "Segment_Format_11_Text_Byte_7" AT %QB611 : Char;
   "Segment_Format_11_Text_Byte_8" AT %QB612 : Char;
   "Segment_Format_11_Text_Byte_9" AT %QB613 : Char;
   "Segment_Format_11_Text_Byte_10" AT %QB614 : Char;
   "Segment_Format_11_Text_Byte_11" AT %QB615 : Char;
   "Segment_Format_11_Text_Byte_12" AT %QB616 : Char;
   "Segment_Format_11_Text_Byte_13" AT %QB617 : Char;
   "Segment_Format_11_Text_Byte_14" AT %QB618 : Char;
   "Segment_Format_11_Text_Byte_15" AT %QB619 : Char;
   "Segment_Format_11_Text_Byte_16" AT %QB620 : Char;
   "Segment_Format_11_Text_Byte_17" AT %QB621 : Char;
   "Segment_Format_11_Text_Byte_18" AT %QB622 : Char;
   "Segment_Format_11_Text_Byte_19" AT %QB623 : Char;
   "Segment_Format_11_Text_Byte_20" AT %QB624 : Char;
   "Segment_Format_11_Text_Byte_21" AT %QB625 : Char;
   "Segment_Format_11_Text_Byte_22" AT %QB626 : Char;
   "Segment_Format_11_Text_Byte_23" AT %QB627 : Char;
   "Segment_Format_11_Text_Byte_24" AT %QB628 : Char;
   "Segment_Format_11_Text_Byte_25" AT %QB629 : Char;
   "Segment_Format_11_Text_Byte_26" AT %QB630 : Char;
   "Segment_Format_11_Text_Byte_27" AT %QB631 : Char;
   "Segment_Format_11_Text_Byte_28" AT %QB632 : Char;
   "Segment_Format_11_Text_Byte_29" AT %QB633 : Char;
   "Segment_Format_11_Text_Byte_30" AT %QB634 : Char;
   "Segment_Format_11_Text_Byte_31" AT %QB635 : Char;
   "Segment_Format_11_Text_Byte_32" AT %QB636 : Char;
   "Segment_Format_11_Text_Byte_33" AT %QB637 : Char;
   "Segment_Format_11_Text_Byte_34" AT %QB638 : Char;
   "Segment_Format_11_Text_Byte_35" AT %QB639 : Char;
   "Segment_Format_11_Text_Byte_36" AT %QB640 : Char;
   "Segment_Format_11_Text_Byte_37" AT %QB641 : Char;
   "Segment_Format_11_Text_Byte_38" AT %QB642 : Char;
   "Segment_Format_11_Text_Byte_39" AT %QB643 : Char;
   "Segment_Format_11_Text_Byte_40" AT %QB644 : Char;
   "Segment_Format_11_Text_Byte_41" AT %QB645 : Char;
   "Segment_Format_11_Text_Byte_42" AT %QB646 : Char;
   "Segment_Format_11_Text_Byte_43" AT %QB647 : Char;
   "Segment_Format_11_Text_Byte_44" AT %QB648 : Char;
   "Segment_Format_11_Text_Byte_45" AT %QB649 : Char;
END_VAR

VAR_GLOBAL   // PLC tag table "Segment Format 12"
   "Segment_Format_12_FG_Color" AT %QB650 : USInt;
   "Segment_Format_12_BG_Color" AT %QB651 : USInt;
   "Segment_Format_12_Flash" AT %QB652 : USInt;
   "Segment_Format_12_Line_Number" AT %QB653 : USInt;
   "Segment_Format_12_Text_Byte_0" AT %QB654 : Char;
   "Segment_Format_12_Text_Byte_1" AT %QB655 : Char;
   "Segment_Format_12_Text_Byte_2" AT %QB656 : Char;
   "Segment_Format_12_Text_Byte_3" AT %QB657 : Char;
   "Segment_Format_12_Text_Byte_4" AT %QB658 : Char;
   "Segment_Format_12_Text_Byte_5" AT %QB659 : Char;
   "Segment_Format_12_Text_Byte_6" AT %QB660 : Char;
   "Segment_Format_12_Text_Byte_7" AT %QB661 : Char;
   "Segment_Format_12_Text_Byte_8" AT %QB662 : Char;
   "Segment_Format_12_Text_Byte_9" AT %QB663 : Char;
   "Segment_Format_12_Text_Byte_10" AT %QB664 : Char;
   "Segment_Format_12_Text_Byte_11" AT %QB665 : Char;
   "Segment_Format_12_Text_Byte_12" AT %QB666 : Char;
   "Segment_Format_12_Text_Byte_13" AT %QB667 : Char;
   "Segment_Format_12_Text_Byte_14" AT %QB668 : Char;
   "Segment_Format_12_Text_Byte_15" AT %QB669 : Char;
   "Segment_Format_12_Text_Byte_16" AT %QB670 : Char;
   "Segment_Format_12_Text_Byte_17" AT %QB671 : Char;
   "Segment_Format_12_Text_Byte_18" AT %QB672 : Char;
   "Segment_Format_12_Text_Byte_19" AT %QB673 : Char;
   "Segment_Format_12_Text_Byte_20" AT %QB674 : Char;
   "Segment_Format_12_Text_Byte_21" AT %QB675 : Char;
   "Segment_Format_12_Text_Byte_22" AT %QB676 : Char;
   "Segment_Format_12_Text_Byte_23" AT %QB677 : Char;
   "Segment_Format_12_Text_Byte_24" AT %QB678 : Char;
   "Segment_Format_12_Text_Byte_25" AT %QB679 : Char;
   "Segment_Format_12_Text_Byte_26" AT %QB680 : Char;
   "Segment_Format_12_Text_Byte_27" AT %QB681 : Char;
   "Segment_Format_12_Text_Byte_28" AT %QB682 : Char;
   "Segment_Format_12_Text_Byte_29" AT %QB683 : Char;
   "Segment_Format_12_Text_Byte_30" AT %QB684 : Char;
   "Segment_Format_12_Text_Byte_31" AT %QB685 : Char;
   "Segment_Format_12_Text_Byte_32" AT %QB686 : Char;
   "Segment_Format_12_Text_Byte_33" AT %QB687 : Char;
   "Segment_Format_12_Text_Byte_34" AT %QB688 : Char;
   "Segment_Format_12_Text_Byte_35" AT %QB689 : Char;
   "Segment_Format_12_Text_Byte_36" AT %QB690 : Char;
   "Segment_Format_12_Text_Byte_37" AT %QB691 : Char;
   "Segment_Format_12_Text_Byte_38" AT %QB692 : Char;
   "Segment_Format_12_Text_Byte_39" AT %QB693 : Char;
   "Segment_Format_12_Text_Byte_40" AT %QB694 : Char;
   "Segment_Format_12_Text_Byte_41" AT %QB695 : Char;
   "Segment_Format_12_Text_Byte_42" AT %QB696 : Char;
   "Segment_Format_12_Text_Byte_43" AT %QB697 : Char;
   "Segment_Format_12_Text_Byte_44" AT %QB698 : Char;
   "Segment_Format_12_Text_Byte_45" AT %QB699 : Char;
END_VAR

VAR_GLOBAL   // PLC tag table "Segment Format 13"
   "Segment_Format_13_FG_Color" AT %QB700 : USInt;
   "Segment_Format_13_BG_Color" AT %QB701 : USInt;
   "Segment_Format_13_Flash" AT %QB702 : USInt;
   "Segment_Format_13_Line_Number" AT %QB703 : USInt;
   "Segment_Format_13_Text_Byte_0" AT %QB704 : Char;
   "Segment_Format_13_Text_Byte_1" AT %QB705 : Char;
   "Segment_Format_13_Text_Byte_2" AT %QB706 : Char;
   "Segment_Format_13_Text_Byte_3" AT %QB707 : Char;
   "Segment_Format_13_Text_Byte_4" AT %QB708 : Char;
   "Segment_Format_13_Text_Byte_5" AT %QB709 : Char;
   "Segment_Format_13_Text_Byte_6" AT %QB710 : Char;
   "Segment_Format_13_Text_Byte_7" AT %QB711 : Char;
   "Segment_Format_13_Text_Byte_8" AT %QB712 : Char;
   "Segment_Format_13_Text_Byte_9" AT %QB713 : Char;
   "Segment_Format_13_Text_Byte_10" AT %QB714 : Char;
   "Segment_Format_13_Text_Byte_11" AT %QB715 : Char;
   "Segment_Format_13_Text_Byte_12" AT %QB716 : Char;
   "Segment_Format_13_Text_Byte_13" AT %QB717 : Char;
   "Segment_Format_13_Text_Byte_14" AT %QB718 : Char;
   "Segment_Format_13_Text_Byte_15" AT %QB719 : Char;
   "Segment_Format_13_Text_Byte_16" AT %QB720 : Char;
   "Segment_Format_13_Text_Byte_17" AT %QB721 : Char;
   "Segment_Format_13_Text_Byte_18" AT %QB722 : Char;
   "Segment_Format_13_Text_Byte_19" AT %QB723 : Char;
   "Segment_Format_13_Text_Byte_20" AT %QB724 : Char;
   "Segment_Format_13_Text_Byte_21" AT %QB725 : Char;
   "Segment_Format_13_Text_Byte_22" AT %QB726 : Char;
   "Segment_Format_13_Text_Byte_23" AT %QB727 : Char;
   "Segment_Format_13_Text_Byte_24" AT %QB728 : Char;
   "Segment_Format_13_Text_Byte_25" AT %QB729 : Char;
   "Segment_Format_13_Text_Byte_26" AT %QB730 : Char;
   "Segment_Format_13_Text_Byte_27" AT %QB731 : Char;
   "Segment_Format_13_Text_Byte_28" AT %QB732 : Char;
   "Segment_Format_13_Text_Byte_29" AT %QB733 : Char;
   "Segment_Format_13_Text_Byte_30" AT %QB734 : Char;
   "Segment_Format_13_Text_Byte_31" AT %QB735 : Char;
   "Segment_Format_13_Text_Byte_32" AT %QB736 : Char;
   "Segment_Format_13_Text_Byte_33" AT %QB737 : Char;
   "Segment_Format_13_Text_Byte_34" AT %QB738 : Char;
   "Segment_Format_13_Text_Byte_35" AT %QB739 : Char;
   "Segment_Format_13_Text_Byte_36" AT %QB740 : Char;
   "Segment_Format_13_Text_Byte_37" AT %QB741 : Char;
   "Segment_Format_13_Text_Byte_38" AT %QB742 : Char;
   "Segment_Format_13_Text_Byte_39" AT %QB743 : Char;
   "Segment_Format_13_Text_Byte_40" AT %QB744 : Char;
   "Segment_Format_13_Text_Byte_41" AT %QB745 : Char;
   "Segment_Format_13_Text_Byte_42" AT %QB746 : Char;
   "Segment_Format_13_Text_Byte_43" AT %QB747 : Char;
   "Segment_Format_13_Text_Byte_44" AT %QB748 : Char;
   "Segment_Format_13_Text_Byte_45" AT %QB749 : Char;
END_VAR

VAR_GLOBAL   // PLC tag table "Segment Format 14"
   "Segment_Format_14_FG_Color" AT %QB750 : USInt;
   "Segment_Format_14_BG_Color" AT %QB751 : USInt;
   "Segment_Format_14_Flash" AT %QB752 : USInt;
   "Segment_Format_14_Line_Number" AT %QB753 : USInt;
   "Segment_Format_14_Text_Byte_0" AT %QB754 : Char;
   "Segment_Format_14_Text_Byte_1" AT %QB755 : Char;
   "Segment_Format_14_Text_Byte_2" AT %QB756 : Char;
   "Segment_Format_14_Text_Byte_3" AT %QB757 : Char;
   "Segment_Format_14_Text_Byte_4" AT %QB758 : Char;
   "Segment_Format_14_Text_Byte_5" AT %QB759 : Char;
   "Segment_Format_14_Text_Byte_6" AT %QB760 : Char;
   "Segment_Format_14_Text_Byte_7" AT %QB761 : Char;
   "Segment_Format_14_Text_Byte_8" AT %QB762 : Char;
   "Segment_Format_14_Text_Byte_9" AT %QB763 : Char;
   "Segment_Format_14_Text_Byte_10" AT %QB764 : Char;
   "Segment_Format_14_Text_Byte_11" AT %QB765 : Char;
   "Segment_Format_14_Text_Byte_12" AT %QB766 : Char;
   "Segment_Format_14_Text_Byte_13" AT %QB767 : Char;
   "Segment_Format_14_Text_Byte_14" AT %QB768 : Char;
   "Segment_Format_14_Text_Byte_15" AT %QB769 : Char;
   "Segment_Format_14_Text_Byte_16" AT %QB770 : Char;
   "Segment_Format_14_Text_Byte_17" AT %QB771 : Char;
   "Segment_Format_14_Text_Byte_18" AT %QB772 : Char;
   "Segment_Format_14_Text_Byte_19" AT %QB773 : Char;
   "Segment_Format_14_Text_Byte_20" AT %QB774 : Char;
   "Segment_Format_14_Text_Byte_21" AT %QB775 : Char;
   "Segment_Format_14_Text_Byte_22" AT %QB776 : Char;
   "Segment_Format_14_Text_Byte_23" AT %QB777 : Char;
   "Segment_Format_14_Text_Byte_24" AT %QB778 : Char;
   "Segment_Format_14_Text_Byte_25" AT %QB779 : Char;
   "Segment_Format_14_Text_Byte_26" AT %QB780 : Char;
   "Segment_Format_14_Text_Byte_27" AT %QB781 : Char;
   "Segment_Format_14_Text_Byte_28" AT %QB782 : Char;
   "Segment_Format_14_Text_Byte_29" AT %QB783 : Char;
   "Segment_Format_14_Text_Byte_30" AT %QB784 : Char;
   "Segment_Format_14_Text_Byte_31" AT %QB785 : Char;
   "Segment_Format_14_Text_Byte_32" AT %QB786 : Char;
   "Segment_Format_14_Text_Byte_33" AT %QB787 : Char;
   "Segment_Format_14_Text_Byte_34" AT %QB788 : Char;
   "Segment_Format_14_Text_Byte_35" AT %QB789 : Char;
   "Segment_Format_14_Text_Byte_36" AT %QB790 : Char;
   "Segment_Format_14_Text_Byte_37" AT %QB791 : Char;
   "Segment_Format_14_Text_Byte_38" AT %QB792 : Char;
   "Segment_Format_14_Text_Byte_39" AT %QB793 : Char;
   "Segment_Format_14_Text_Byte_40" AT %QB794 : Char;
   "Segment_Format_14_Text_Byte_41" AT %QB795 : Char;
   "Segment_Format_14_Text_Byte_42" AT %QB796 : Char;
   "Segment_Format_14_Text_Byte_43" AT %QB797 : Char;
   "Segment_Format_14_Text_Byte_44" AT %QB798 : Char;
   "Segment_Format_14_Text_Byte_45" AT %QB799 : Char;
END_VAR

VAR_GLOBAL   // PLC tag table "Segment Format 15"
   "Segment_Format_15_FG_Color" AT %QB800 : USInt;
   "Segment_Format_15_BG_Color" AT %QB801 : USInt;
   "Segment_Format_15_Flash" AT %QB802 : USInt;
   "Segment_Format_15_Line_Number" AT %QB803 : USInt;
   "Segment_Format_15_Text_Byte_0" AT %QB804 : Char;
   "Segment_Format_15_Text_Byte_1" AT %QB805 : Char;
   "Segment_Format_15_Text_Byte_2" AT %QB806 : Char;
   "Segment_Format_15_Text_Byte_3" AT %QB807 : Char;
   "Segment_Format_15_Text_Byte_4" AT %QB808 : Char;
   "Segment_Format_15_Text_Byte_5" AT %QB809 : Char;
   "Segment_Format_15_Text_Byte_6" AT %QB810 : Char;
   "Segment_Format_15_Text_Byte_7" AT %QB811 : Char;
   "Segment_Format_15_Text_Byte_8" AT %QB812 : Char;
   "Segment_Format_15_Text_Byte_9" AT %QB813 : Char;
   "Segment_Format_15_Text_Byte_10" AT %QB814 : Char;
   "Segment_Format_15_Text_Byte_11" AT %QB815 : Char;
   "Segment_Format_15_Text_Byte_12" AT %QB816 : Char;
   "Segment_Format_15_Text_Byte_13" AT %QB817 : Char;
   "Segment_Format_15_Text_Byte_14" AT %QB818 : Char;
   "Segment_Format_15_Text_Byte_15" AT %QB819 : Char;
   "Segment_Format_15_Text_Byte_16" AT %QB820 : Char;
   "Segment_Format_15_Text_Byte_17" AT %QB821 : Char;
   "Segment_Format_15_Text_Byte_18" AT %QB822 : Char;
   "Segment_Format_15_Text_Byte_19" AT %QB823 : Char;
   "Segment_Format_15_Text_Byte_20" AT %QB824 : Char;
   "Segment_Format_15_Text_Byte_21" AT %QB825 : Char;
   "Segment_Format_15_Text_Byte_22" AT %QB826 : Char;
   "Segment_Format_15_Text_Byte_23" AT %QB827 : Char;
   "Segment_Format_15_Text_Byte_24" AT %QB828 : Char;
   "Segment_Format_15_Text_Byte_25" AT %QB829 : Char;
   "Segment_Format_15_Text_Byte_26" AT %QB830 : Char;
   "Segment_Format_15_Text_Byte_27" AT %QB831 : Char;
   "Segment_Format_15_Text_Byte_28" AT %QB832 : Char;
   "Segment_Format_15_Text_Byte_29" AT %QB833 : Char;
   "Segment_Format_15_Text_Byte_30" AT %QB834 : Char;
   "Segment_Format_15_Text_Byte_31" AT %QB835 : Char;
   "Segment_Format_15_Text_Byte_32" AT %QB836 : Char;
   "Segment_Format_15_Text_Byte_33" AT %QB837 : Char;
   "Segment_Format_15_Text_Byte_34" AT %QB838 : Char;
   "Segment_Format_15_Text_Byte_35" AT %QB839 : Char;
   "Segment_Format_15_Text_Byte_36" AT %QB840 : Char;
   "Segment_Format_15_Text_Byte_37" AT %QB841 : Char;
   "Segment_Format_15_Text_Byte_38" AT %QB842 : Char;
   "Segment_Format_15_Text_Byte_39" AT %QB843 : Char;
   "Segment_Format_15_Text_Byte_40" AT %QB844 : Char;
   "Segment_Format_15_Text_Byte_41" AT %QB845 : Char;
   "Segment_Format_15_Text_Byte_42" AT %QB846 : Char;
   "Segment_Format_15_Text_Byte_43" AT %QB847 : Char;
   "Segment_Format_15_Text_Byte_44" AT %QB848 : Char;
   "Segment_Format_15_Text_Byte_45" AT %QB849 : Char;
END_VAR

VAR_GLOBAL   // PLC tag table "Segment Format 16"
   "Segment_Format_16_FG_Color" AT %QB850 : USInt;
   "Segment_Format_16_BG_Color" AT %QB851 : USInt;
   "Segment_Format_16_Flash" AT %QB852 : USInt;
   "Segment_Format_16_Line_Number" AT %QB853 : USInt;
   "Segment_Format_16_Text_Byte_0" AT %QB854 : Char;
   "Segment_Format_16_Text_Byte_1" AT %QB855 : Char;
   "Segment_Format_16_Text_Byte_2" AT %QB856 : Char;
   "Segment_Format_16_Text_Byte_3" AT %QB857 : Char;
   "Segment_Format_16_Text_Byte_4" AT %QB858 : Char;
   "Segment_Format_16_Text_Byte_5" AT %QB859 : Char;
   "Segment_Format_16_Text_Byte_6" AT %QB860 : Char;
   "Segment_Format_16_Text_Byte_7" AT %QB861 : Char;
   "Segment_Format_16_Text_Byte_8" AT %QB862 : Char;
   "Segment_Format_16_Text_Byte_9" AT %QB863 : Char;
   "Segment_Format_16_Text_Byte_10" AT %QB864 : Char;
   "Segment_Format_16_Text_Byte_11" AT %QB865 : Char;
   "Segment_Format_16_Text_Byte_12" AT %QB866 : Char;
   "Segment_Format_16_Text_Byte_13" AT %QB867 : Char;
   "Segment_Format_16_Text_Byte_14" AT %QB868 : Char;
   "Segment_Format_16_Text_Byte_15" AT %QB869 : Char;
   "Segment_Format_16_Text_Byte_16" AT %QB870 : Char;
   "Segment_Format_16_Text_Byte_17" AT %QB871 : Char;
   "Segment_Format_16_Text_Byte_18" AT %QB872 : Char;
   "Segment_Format_16_Text_Byte_19" AT %QB873 : Char;
   "Segment_Format_16_Text_Byte_20" AT %QB874 : Char;
   "Segment_Format_16_Text_Byte_21" AT %QB875 : Char;
   "Segment_Format_16_Text_Byte_22" AT %QB876 : Char;
   "Segment_Format_16_Text_Byte_23" AT %QB877 : Char;
   "Segment_Format_16_Text_Byte_24" AT %QB878 : Char;
   "Segment_Format_16_Text_Byte_25" AT %QB879 : Char;
   "Segment_Format_16_Text_Byte_26" AT %QB880 : Char;
   "Segment_Format_16_Text_Byte_27" AT %QB881 : Char;
   "Segment_Format_16_Text_Byte_28" AT %QB882 : Char;
   "Segment_Format_16_Text_Byte_29" AT %QB883 : Char;
   "Segment_Format_16_Text_Byte_30" AT %QB884 : Char;
   "Segment_Format_16_Text_Byte_31" AT %QB885 : Char;
   "Segment_Format_16_Text_Byte_32" AT %QB886 : Char;
   "Segment_Format_16_Text_Byte_33" AT %QB887 : Char;
   "Segment_Format_16_Text_Byte_34" AT %QB888 : Char;
   "Segment_Format_16_Text_Byte_35" AT %QB889 : Char;
   "Segment_Format_16_Text_Byte_36" AT %QB890 : Char;
   "Segment_Format_16_Text_Byte_37" AT %QB891 : Char;
   "Segment_Format_16_Text_Byte_38" AT %QB892 : Char;
   "Segment_Format_16_Text_Byte_39" AT %QB893 : Char;
   "Segment_Format_16_Text_Byte_40" AT %QB894 : Char;
   "Segment_Format_16_Text_Byte_41" AT %QB895 : Char;
   "Segment_Format_16_Text_Byte_42" AT %QB896 : Char;
   "Segment_Format_16_Text_Byte_43" AT %QB897 : Char;
   "Segment_Format_16_Text_Byte_44" AT %QB898 : Char;
   "Segment_Format_16_Text_Byte_45" AT %QB899 : Char;
END_VAR

VAR_GLOBAL   // PLC tag table "Segment Format 17"
   "Segment_Format_17_FG_Color" AT %QB900 : USInt;
   "Segment_Format_17_BG_Color" AT %QB901 : USInt;
   "Segment_Format_17_Flash" AT %QB902 : USInt;
   "Segment_Format_17_Line_Number" AT %QB903 : USInt;
   "Segment_Format_17_Text_Byte_0" AT %QB904 : Char;
   "Segment_Format_17_Text_Byte_1" AT %QB905 : Char;
   "Segment_Format_17_Text_Byte_2" AT %QB906 : Char;
   "Segment_Format_17_Text_Byte_3" AT %QB907 : Char;
   "Segment_Format_17_Text_Byte_4" AT %QB908 : Char;
   "Segment_Format_17_Text_Byte_5" AT %QB909 : Char;
   "Segment_Format_17_Text_Byte_6" AT %QB910 : Char;
   "Segment_Format_17_Text_Byte_7" AT %QB911 : Char;
   "Segment_Format_17_Text_Byte_8" AT %QB912 : Char;
   "Segment_Format_17_Text_Byte_9" AT %QB913 : Char;
   "Segment_Format_17_Text_Byte_10" AT %QB914 : Char;
   "Segment_Format_17_Text_Byte_11" AT %QB915 : Char;
   "Segment_Format_17_Text_Byte_12" AT %QB916 : Char;
   "Segment_Format_17_Text_Byte_13" AT %QB917 : Char;
   "Segment_Format_17_Text_Byte_14" AT %QB918 : Char;
   "Segment_Format_17_Text_Byte_15" AT %QB919 : Char;
   "Segment_Format_17_Text_Byte_16" AT %QB920 : Char;
   "Segment_Format_17_Text_Byte_17" AT %QB921 : Char;
   "Segment_Format_17_Text_Byte_18" AT %QB922 : Char;
   "Segment_Format_17_Text_Byte_19" AT %QB923 : Char;
   "Segment_Format_17_Text_Byte_20" AT %QB924 : Char;
   "Segment_Format_17_Text_Byte_21" AT %QB925 : Char;
   "Segment_Format_17_Text_Byte_22" AT %QB926 : Char;
   "Segment_Format_17_Text_Byte_23" AT %QB927 : Char;
   "Segment_Format_17_Text_Byte_24" AT %QB928 : Char;
   "Segment_Format_17_Text_Byte_25" AT %QB929 : Char;
   "Segment_Format_17_Text_Byte_26" AT %QB930 : Char;
   "Segment_Format_17_Text_Byte_27" AT %QB931 : Char;
   "Segment_Format_17_Text_Byte_28" AT %QB932 : Char;
   "Segment_Format_17_Text_Byte_29" AT %QB933 : Char;
   "Segment_Format_17_Text_Byte_30" AT %QB934 : Char;
   "Segment_Format_17_Text_Byte_31" AT %QB935 : Char;
   "Segment_Format_17_Text_Byte_32" AT %QB936 : Char;
   "Segment_Format_17_Text_Byte_33" AT %QB937 : Char;
   "Segment_Format_17_Text_Byte_34" AT %QB938 : Char;
   "Segment_Format_17_Text_Byte_35" AT %QB939 : Char;
   "Segment_Format_17_Text_Byte_36" AT %QB940 : Char;
   "Segment_Format_17_Text_Byte_37" AT %QB941 : Char;
   "Segment_Format_17_Text_Byte_38" AT %QB942 : Char;
   "Segment_Format_17_Text_Byte_39" AT %QB943 : Char;
   "Segment_Format_17_Text_Byte_40" AT %QB944 : Char;
   "Segment_Format_17_Text_Byte_41" AT %QB945 : Char;
   "Segment_Format_17_Text_Byte_42" AT %QB946 : Char;
   "Segment_Format_17_Text_Byte_43" AT %QB947 : Char;
   "Segment_Format_17_Text_Byte_44" AT %QB948 : Char;
   "Segment_Format_17_Text_Byte_45" AT %QB949 : Char;
END_VAR

VAR_GLOBAL CONSTANT   // PLC tag table "Constants"
   "LED_NORMAL_5" : SInt := 1;
   "LED_NORMAL_7" : SInt := 2;
   "LED_NORMAL_9" : SInt := 3;
   "LED_NORMAL_11" : SInt := 4;
   "LED_NORMAL_14" : SInt := 5;
   "LED_NORMAL_15" : SInt := 6;
   "LED_NORMAL_16" : SInt := 7;
   "LED_NORMAL_22" : SInt := 8;
   "LED_NORMAL_24" : SInt := 9;
   "LED_NORMAL_30" : SInt := 10;
   "LED_NORMAL_32" : SInt := 11;
   "LED_NORMAL_40" : SInt := 12;
   "LED_BOLD_5" : SInt := 13;
   "LED_BOLD_11" : SInt := 14;
   "LED_BOLD_14" : SInt := 15;
   "LED_BOLD_15" : SInt := 16;
   "LED_BOLD_16" : SInt := 17;
   "LED_BOLD_22" : SInt := 18;
   "LED_BOLD_30" : SInt := 19;
   "LED_BOLD_32" : SInt := 20;
   "LED_BOLD_40" : SInt := 21;
   "LED_SCROLL_FASTEST" : SInt := 1;
   "LED_SCROLL_FAST" : SInt := 2;
   "LED_SCROLL_NORMAL" : SInt := 3;
   "LED_SCROLL_SLOW" : SInt := 4;
   "LED_SCROLL_SLOWEST" : SInt := 5;
   "LED_LEFT" : SInt := 1;
   "LED_CENTER" : SInt := 2;
   "LED_RIGHT" : SInt := 3;
   "LED_HOLD_BOTTOM" : SInt := 1;
   "LED_HOLD_FILL" : SInt := 2;
   "LED_HOLD_MIDDLE" : SInt := 3;
   "LED_HOLD_TOP" : SInt := 4;
   "LED_SCROLL_BOTTOM" : SInt := 5;
   "LED_SCROLL_FILL" : SInt := 6;
   "LED_SCROLL_MIDDLE" : SInt := 7;
   "LED_SCROLL_TOP" : SInt := 8;
   "LED_BLACK" : SInt := 1;
   "LED_RED" : SInt := 2;
   "LED_GREEN" : SInt := 3;
   "LED_YELLOW" : SInt := 4;
   "LED_MIX_1" : SInt := 5;
   "LED_MIX_2" : SInt := 6;
   "LED_MIX_3" : SInt := 7;
   "LED_MIX_4" : SInt := 8;
   "LED_BLUE" : SInt := 9;
   "LED_WHITE" : SInt := 10;
   "LED_FLASH_ON" : SInt := 1;
   "LED_FLASH_OFF" : SInt := 2;
END_VAR

VAR_GLOBAL   // PLC tag table "System Parameters"
   "IP_1" AT %QB0 : USInt;
   "IP_2" AT %QB1 : USInt;
   "IP_3" AT %QB2 : USInt;
   "IP_4" AT %QB3 : USInt;
   "PORT_MSB" AT %QB4 : Byte;
   "PORT_LSB" AT %QB5 : Byte;
   "REQUESTS" AT %QB6 : Byte;
END_VAR

VAR_GLOBAL   // PLC tag table "Sign Format"
   "Hold" AT %QB10 : USInt;
   "Scroll_Speed" AT %QB11 : USInt;
   "Vertical_Alignment" AT %QB12 : USInt;
END_VAR

// folder: ADP Gateway Interface

TYPE "ADP_Gateway_Interface.UDT"
   STRUCT
      hardware_address : DInt;
      line_format : Array[0..4] of "ADP_Gateway_Interface.Line_Format.UDT";
      sign_format : "ADP_Gateway_Interface.Sign_Format.UDT";
      segment_format : Array[0..17] of "ADP_Gateway_Interface.Segment_Format.UDT";
      system_parameters : "ADP_Gateway_Interface.System_Parameters.UDT";
   END_STRUCT;
END_TYPE

TYPE "ADP_Gateway_Interface.Line_Format.UDT"
   STRUCT
      font : SInt := 1;
      horizontal_alignment : SInt := 1;
   END_STRUCT;
END_TYPE

TYPE "ADP_Gateway_Interface.Segment_Format.UDT"
   STRUCT
      foreground_color : SInt := 1;
      background_color : SInt := 1;
      flash : SInt := 1;
      line_number : SInt := -1;
      text : String[46];
   END_STRUCT;
END_TYPE

TYPE "ADP_Gateway_Interface.System_Parameters.UDT"
   STRUCT
      ip_address : String[15];
      port : String[5];
      reset_request : Bool;
   END_STRUCT;
END_TYPE

TYPE "ADP_Gateway_Interface.Sign_Format.UDT"
   STRUCT
      hold : SInt := 5;
      scroll_speed : SInt := 1;
      vertical_alignment : SInt := 1;
   END_STRUCT;
END_TYPE

// folder: (top level)

DATA_BLOCK "DEBUG"   // DB2
{ S7_Optimized_Access := 'TRUE' }
VERSION : 0.1
   VAR
      count : UDInt;
      clock : Bool;
      clock_memory : Bool;
   END_VAR
BEGIN
END_DATA_BLOCK

// folder: ADP Gateway Interface

DATA_BLOCK "ADP_Gateway_Interface.Data"   // DB1
{ S7_Optimized_Access := 'TRUE' }
VERSION : 0.1
BEGIN
END_DATA_BLOCK

// folder: (top level)

FUNCTION "String.trim" : String   // FC12, SCL
{ S7_Optimized_Access := 'TRUE' }
AUTHOR : Machado
FAMILY : String
VERSION : 1.0
// removes leading and trailing whitespace from input string
   VAR_INPUT
      "string" : String;
   END_VAR
   VAR_TEMP
      ret : String;
   END_VAR
   VAR CONSTANT
      space : String := ' ';
   END_VAR
BEGIN
   #ret := #string;
   WHILE LEFT(IN := #ret, L := 1) = #space DO
       #ret := RIGHT(IN := #ret, L := LEN(#ret) - 1);
   END_WHILE;
   WHILE RIGHT(IN := #ret, L := 1) = #space DO
       #ret := LEFT(IN := #ret, L := LEN(#ret) - 1);
   END_WHILE;
   #"String.trim" := #ret;
END_FUNCTION

ORGANIZATION_BLOCK "Main"   // OB1, LAD, ProgramCycle
TITLE = "Main Program Sweep (Cycle)"
{ S7_Optimized_Access := 'TRUE' }
VERSION : 0.1
   VAR_INPUT
      Initial_Call : Bool;   // Initial call of this OB
      Remanence : Bool;   // =True, if remanent data are available
   END_VAR
BEGIN

REGION Network 1
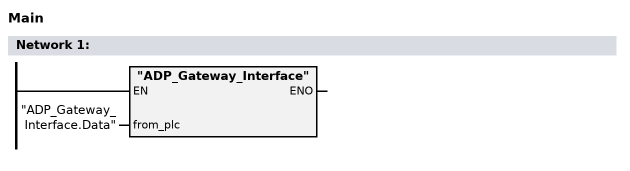
   RUNG wire#powerrail
      "ADP_Gateway_Interface"(from_plc := "ADP_Gateway_Interface.Data")
   END_RUNG
   // the same network as SCL:
   "ADP_Gateway_Interface"(from_plc := "ADP_Gateway_Interface.Data");
END_REGION

REGION Network 2 (SCL)
   "DEBUG".clock := "Clock_2Hz";
   IF "DEBUG".clock AND NOT "DEBUG".clock_memory THEN
       "DEBUG".count += 1;
   END_IF;
   IF "DEBUG".count = 999999 THEN
       "DEBUG".count := 0;
   END_IF;
   "DEBUG".clock_memory := "DEBUG".clock;
   "ADP_Gateway_Interface.Data".segment_format[0].text := '';
   "ADP_Gateway_Interface.Data".segment_format[0].text := "String.trim"(UDINT_TO_STRING("DEBUG".count));
END_REGION
END_ORGANIZATION_BLOCK

// folder: ADP Gateway Interface

FUNCTION "ADP_Gateway_Interface" : Void   // FC1, SCL
TITLE = ADP Gateway Interface
{ S7_Optimized_Access := 'TRUE' }
AUTHOR : Machado
VERSION : 0.1
// for use with GSD file version xxxxx
   VAR_INPUT
      from_plc : "ADP_Gateway_Interface.UDT";
   END_VAR
   VAR_TEMP
      i : DInt;
      ip_as_string : String;
      j : DInt;
      octet_as_byte : Byte;
      octet_as_dint : DInt;
      octet_as_string : String;
      offset : DInt;
      port_as_dint : DInt;
      port_as_uint : UInt;
      position : Int;
      requests_as_byte : Byte;
   END_VAR
   VAR CONSTANT
      FORMAT : Word;
      LINE_COUNT : DInt := 4;   // 5 lines, 0 indexed
      NO_DB : DInt;
      OUTPUT_AREA : Byte := 16#82;
      SEGMENT_FORMAT_COUNT : DInt := 17;   // 18 format segments, 0 indexed
      SYSTEM_PARAMETERS_AREA_START : DInt := 0;
      SIGN_FORMAT_AREA_START : DInt := 10;
      LINE_FORMAT_AREA_START : DInt := 20;
      SEGMENT_FORMAT_AREA_START : DInt := 50;
      TEXT_CHARACTER_COUNT : DInt := 46;   // 1 indexed
   END_VAR
BEGIN
   REGION "SYSTEM PARAMETERS"

       REGION "INITIALIZE OFFSET"
           #offset := #from_plc.hardware_address + #SYSTEM_PARAMETERS_AREA_START;
       END_REGION

       REGION "POKE IP ADDRESS"
           // INITIALIZE LOCALS
           #ip_as_string := #from_plc.system_parameters.ip_address;
           #i := 0;
           // LOOP THROUGH OCTETS OF IP ADDRESS
           WHILE LEN(#ip_as_string) > 0 DO
               // GET POSITION OF DELIMETER (PERIOD IN IP ADDRESS)
               #position := FIND(IN1 := #ip_as_string,
                                 IN2 := '.');
               // DELIMETER NOT FOUND
               IF #position <= 0 THEN
                   #octet_as_string := #ip_as_string;
                   #ip_as_string := '';
               END_IF;
               // DELIMETER FOUND
               IF #position > 0 THEN
                   #octet_as_string := LEFT_STRING(IN := #ip_as_string,
                                                   L := #position - 1);
                   #ip_as_string := RIGHT_STRING(IN := #ip_as_string,
                                                 L := LEN(#ip_as_string) - #position);
               END_IF;
               // CONVERT STRING OCTET TO BYTE OCTET
               STRG_VAL(IN := #octet_as_string,
                        FORMAT := #FORMAT,
                        P := 1,
                        OUT => #octet_as_dint);
               IF #octet_as_dint < 0 OR #octet_as_dint > 255 THEN
                   #octet_as_dint := 0;
               END_IF;
               #octet_as_byte := DINT_TO_BYTE(#octet_as_dint);
               // WRITE OCTET TO OUTPUT AREA
               POKE(area := #OUTPUT_AREA,
                    dbNumber := #NO_DB,
                    byteOffset := #offset,
                    value := #octet_as_byte);
               #offset += 1;
           END_WHILE;
       END_REGION

       REGION "POKE PORT"
           STRG_VAL(IN := #from_plc.system_parameters."port",
               FORMAT := #FORMAT,
               P := 1,
               OUT => #port_as_dint);
           #port_as_uint := DINT_TO_UINT(#port_as_dint);
           POKE(area := #OUTPUT_AREA,
                dbNumber := #NO_DB,
                byteOffset := #offset,
                value := #port_as_uint.%B0);
           #offset += 1;
           POKE(area := #OUTPUT_AREA,
                dbNumber := #NO_DB,
                byteOffset := #offset,
                value := #port_as_uint.%B1);
           #offset += 1;
       END_REGION

       REGION "POKE REQUESTS"
           #requests_as_byte.%X0 := #from_plc.system_parameters.reset_request;
           POKE(area := #OUTPUT_AREA,
                dbNumber := #NO_DB,
                byteOffset := #offset,
                value := #requests_as_byte);
           #offset += 1;
       END_REGION

   END_REGION


   REGION "SIGN FORMATS"

       REGION "INITIALIZE OFFSET"
           #offset := #from_plc.hardware_address + #SIGN_FORMAT_AREA_START;
       END_REGION

       REGION "HOLD"
           POKE(area := #OUTPUT_AREA,
                dbNumber := #NO_DB,
                byteOffset := #offset,
                value := SINT_TO_BYTE(#from_plc.sign_format.hold));
           #offset += 1;
       END_REGION

       REGION "SCROLL SPEED"
           POKE(area := #OUTPUT_AREA,
                dbNumber := #NO_DB,
                byteOffset := #offset,
                value := SINT_TO_BYTE(#from_plc.sign_format.scroll_speed));
           #offset += 1;
       END_REGION

       REGION "VERTICAL ALIGNMENT"
           POKE(area := #OUTPUT_AREA,
                dbNumber := #NO_DB,
                byteOffset := #offset,
                value := SINT_TO_BYTE(#from_plc.sign_format.vertical_alignment));
           #offset += 1;
       END_REGION

   END_REGION


   REGION "LINE FORMATS"

       REGION "INITIALIZE OFFSET"
           #offset := #from_plc.hardware_address + #LINE_FORMAT_AREA_START;
       END_REGION

       REGION "LOOP THROUGH LINES"
           FOR #i := 0 TO #LINE_COUNT DO

               REGION "FONT"
                   POKE(area := #OUTPUT_AREA,
                        dbNumber := #NO_DB,
                        byteOffset := #offset,
                        value := SINT_TO_BYTE(#from_plc.line_format[#i].font));
                   #offset += 1;
               END_REGION

               REGION "VERTICAL ALIGNMENT"
                   POKE(area := #OUTPUT_AREA,
                        dbNumber := #NO_DB,
                        byteOffset := #offset,
                        value := SINT_TO_BYTE(#from_plc.line_format[#i].horizontal_alignment));
                   #offset += 1;
               END_REGION

           END_FOR;
       END_REGION

   END_REGION


   REGION "SEGMENT FORMATS"

       REGION "INITIALIZE OFFSET"
           #offset := #from_plc.hardware_address + #SEGMENT_FORMAT_AREA_START;
       END_REGION

       REGION "LOOP THROUGH SEGMENT FORMATS"
           FOR #i := 0 TO #SEGMENT_FORMAT_COUNT DO

               REGION "FOREGROUND COLOR"
                   POKE(area := #OUTPUT_AREA,
                        dbNumber := #NO_DB,
                        byteOffset := #offset,
                        value := SINT_TO_BYTE(#from_plc.segment_format[#i].foreground_color));
                   #offset += 1;
               END_REGION

               REGION "BACKGROUND COLOR"
                   POKE(area := #OUTPUT_AREA,
                        dbNumber := #NO_DB,
                        byteOffset := #offset,
                        value := SINT_TO_BYTE(#from_plc.segment_format[#i].background_color));
                   #offset += 1;
               END_REGION

               REGION "FLASH"
                   POKE(area := #OUTPUT_AREA,
                        dbNumber := #NO_DB,
                        byteOffset := #offset,
                        value := SINT_TO_BYTE(#from_plc.segment_format[#i].flash));
                   #offset += 1;
               END_REGION

               REGION "LINE NUMBER"
                   POKE(area := #OUTPUT_AREA,
                        dbNumber := #NO_DB,
                        byteOffset := #offset,
                        value := SINT_TO_BYTE(#from_plc.segment_format[#i].line_number));
                   #offset += 1;
               END_REGION

               REGION "TEXT"
                   FOR #j := 1 TO #TEXT_CHARACTER_COUNT DO
                       POKE(area := #OUTPUT_AREA,
                            dbNumber := #NO_DB,
                            byteOffset := #offset,
                            value := CHAR_TO_BYTE(#from_plc.segment_format[#i].text[#j]));
                       #offset += 1;
                   END_FOR;
               END_REGION

           END_FOR;
       END_REGION

   END_REGION


   REGION "RETURN"
       #offset := #offset;
       RETURN;
   END_REGION
END_FUNCTION